FUNCTION_BLOCK FINAL FB_Diagnostics EXTENDS FB_EventLogger 
VAR_IN_OUT
	Control				: ST_System;					  //Machine Control Instance
	Trigger				: BOOL;							  //Diagnostic function call interval
END_VAR
VAR_OUTPUT
	ncpuUsage 			: UDINT;						  //CPU Usage
	nlatency 			: UDINT;						  //CPU Latency
	Outputs 			: ARRAY[0..255] OF ST_Diagnostics;//Devices on ECAT Bus
	ControllerID		: ST_DeviceIdentificationEx;	  //IPC Information
	IPAddress			: T_IPv4Addr;					  //IPC ip address
END_VAR                                                   
VAR                                                       
	_Alarm				: BOOL;							  //Device Alarm
	_AlarmNum			: DINT;							  //Device Alarm Number
	_Warning			: BOOL;							  //Device Warning
	_WarningNum			: DINT;							  //Device Warning Number
	_FaultTimer_ET		: REAL;								//Fault timer elapsed
	_r_Trig				: ARRAY[0..9] OF R_TRIG;    	  //Public Rising Edge Triggers
END_VAR                                                   
VAR_STAT                                                  
	_Masterdata			: ARRAY[0..10] OF ST_Masterdata;  //ECAT Master Device Diagnostic Data
	_DeviceFault		: BOOL;							  //Fault for crc count
	_StatusFault		: BOOL;							  //Fault for status
END_VAR
VAR PERSISTENT          	
	_Name					: STRING[40];				  //Name for HMI
	_Description			: STRING[40];				  //Description for HMI
	_AlarmMute				: BOOL;						  //Alarm Mute
	_FaultTimer_PT			: REAL;						  //Fault timer preset time
END_VAR

M_CPU();
M_Masters();
M_Slaves();
M_AlarmMonitor();
M_AlarmReset();
M_WarningMonitor();

{attribute 'monitoring' := 'variable'}
PROPERTY PUBLIC Alarm : Bool
GET
Alarm := _Alarm;
END_GET
END_PROPERTY

{attribute 'monitoring' := 'variable'}
PROPERTY PUBLIC AlarmMute : BOOL
SET
AlarmMute := _AlarmMute;
END_SET
END_PROPERTY

{attribute 'monitoring' := 'variable'}
PROPERTY PUBLIC Description : String[40]
GET
Description := _Description;
END_GET
SET
_Description := Description;
END_SET
END_PROPERTY

METHOD PRIVATE F_DeviceState_to_String : STRING
VAR_INPUT
	DeviceState: BYTE;
END_VAR
CASE (DeviceState AND 16#0F) OF
	1: F_DeviceState_to_String := 'Init';
	2: F_DeviceState_to_String := 'Pre-Operational';
	3: F_DeviceState_to_String := 'Bootstrap';
	4: F_DeviceState_to_String := 'Safe-Operational';
	8: F_DeviceState_to_String := 'Operational'; 
END_CASE
CASE (DeviceState AND 16#F0) OF
	1: F_DeviceState_to_String := Concat(F_DeviceState_to_String,': Statemachine error in the EtherCAT slave');
	2: F_DeviceState_to_String := Concat(F_DeviceState_to_String,': Invalid VendorId, Product Code, RevisionsNo or SerialNo');
	4: F_DeviceState_to_String := Concat(F_DeviceState_to_String,': Error occured while sending initialization commands.');
END_CASE
RETURN;
END_METHOD

METHOD PRIVATE F_LinkState_to_String : STRING
VAR_INPUT
	LinkState: BYTE;
END_VAR
CASE (LinkState AND 16#0F) OF
	0: F_LinkState_to_String := 'Link status ok';
	1: F_LinkState_to_String := 'No communication with the EtherCAT-Slave';
	2: F_LinkState_to_String := concat(concat('Error at port ', INT_TO_STRING(((LinkState AND 16#F0)/16)-1)), '. The port has a link, but no communication is possible.');
	4: F_LinkState_to_String := concat(concat('Missing link at port ', BYTE_TO_STRING(((LinkState AND 16#F0)/16)-1)), '.');
	8: F_LinkState_to_String := concat(concat('Additional link at port ', BYTE_TO_STRING(((LinkState AND 16#F0)/16)-1)), '.'); 
END_CASE
RETURN;
END_METHOD

{attribute 'monitoring' := 'variable'}
PROPERTY PUBLIC FaultTimer_PT : real
GET
FaultTimer_PT := _FaultTimer_PT;
END_GET
SET
_FaultTimer_PT := FaultTimer_PT;
END_SET
END_PROPERTY

METHOD PRIVATE M_AlarmMonitor
VAR
END_VAR
VAR_INST // added by the converter: edge detectors and wires of the graphical bodies
    _w1, _w2, _w3, _w4, _w5 : BOOL;
END_VAR
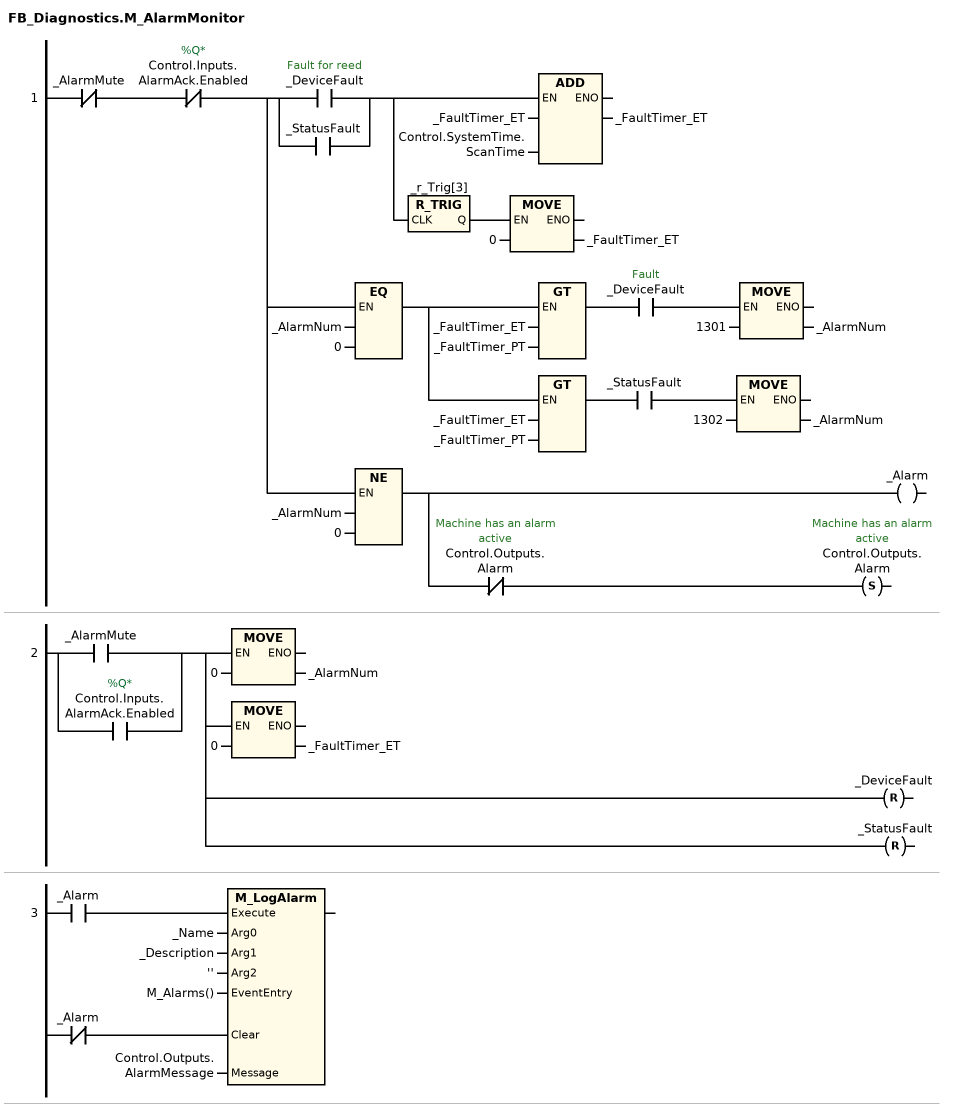
// NETWORK 1
//   Control.Inputs.AlarmAck.Enabled: AT %Q*
//   _DeviceFault: Fault
//   _FaultTimer_ET: Fault timer elapsed
//   Control.SystemTime.ScanTime: Last scan time (Seconds)
//   _FaultTimer_PT: Fault timer preset time
//   Control.Outputs.Alarm: Machine has an alarm active
_w1 := NOT _AlarmMute AND NOT Control.Inputs.AlarmAck.Enabled;
_w2 := _w1 AND (_DeviceFault OR _StatusFault);
IF _w2 THEN _FaultTimer_ET := _FaultTimer_ET + Control.SystemTime.ScanTime; END_IF
_r_Trig[3](CLK := _w2); // R_TRIG
IF _r_Trig[3].Q THEN _FaultTimer_ET := 0; END_IF
_w3 := _w1 AND _AlarmNum = 0;
IF (_w3 AND _FaultTimer_ET > _FaultTimer_PT) AND _DeviceFault THEN _AlarmNum := 1301; END_IF
IF (_w3 AND _FaultTimer_ET > _FaultTimer_PT) AND _StatusFault THEN _AlarmNum := 1302; END_IF
_w4 := _w1 AND _AlarmNum <> 0;
_Alarm := _w4;
Control.Outputs.Alarm S= _w4 AND NOT Control.Outputs.Alarm;

// NETWORK 2
//   Control.Inputs.AlarmAck.Enabled: AT %Q*
//   _FaultTimer_ET: Fault timer elapsed
_w5 := _AlarmMute OR Control.Inputs.AlarmAck.Enabled;
IF _w5 THEN _AlarmNum := 0; END_IF
IF _w5 THEN _FaultTimer_ET := 0; END_IF
_DeviceFault R= _w5;
_StatusFault R= _w5;

// NETWORK 3
M_LogAlarm(Execute := _Alarm, Arg0 := _Name, Arg1 := _Description, Arg2 := '', EventEntry := M_Alarms(), Clear := NOT _Alarm, Message := Control.Outputs.AlarmMessage);
END_METHOD

METHOD PRIVATE M_AlarmReset
VAR_STAT	
	_ClearCRC			:FB_EcMasterFrameStatisticClearCRC; 
	_ClearFrames		:FB_EcMasterFrameStatisticClearFrames;
	_step				: INT;
	_counter			: INT;
END_VAR
// Step engine for resetting etherCat mater errors

CASE _step OF
	0 :	// Initialise and wait for trigger
		_ClearCRC.bExecute:=FALSE;
		_ClearFrames.bExecute:=FALSE;
		_counter := 0;
		IF Control.Inputs.AlarmAck.Enabled THEN _step:=_step+1; END_IF

	
	1 :	// Start getting device ID's 
		_ClearCRC.sNetId := _Masterdata[_counter].NetId;
		_ClearCRC.bExecute:=TRUE;
		IF _ClearCRC.bBusy OR _ClearCRC.bError THEN
		_step:=_step+1; END_IF

	
	2 :	// Getting ID's complete
		_ClearCRC.bExecute:=FALSE;
		IF NOT _ClearCRC.bBusy THEN
		_step:=_step+1;END_IF

	
	3 :	// Start getting device name from device ID
		_ClearFrames.sNetId := _Masterdata[_counter].NetId;
		_ClearFrames.bExecute:=TRUE;
		IF _ClearFrames.bBusy OR _ClearFrames.bError THEN
		_step:=_step+1;END_IF

	
	4 :	// Getting device name complete
		_ClearFrames.bExecute:=FALSE;
		IF NOT _ClearFrames.bBusy THEN
		_step:=_step+1;END_IF

		
	5 :	// Start getting device AMS Net ID from device ID
		_counter := _counter + 1;
		IF _counter >= 11 THEN
		_step:=0;ELSE
		_step:=1;END_IF
			
ELSE
	_step:=0;
END_CASE

// Function block calls
_ClearCRC(sNetId:=);
_ClearFrames(sNetId:=);
END_METHOD

METHOD M_Alarms : TcEventEntry
VAR_INPUT
END_VAR
CASE _AlarmNum OF
	1301: M_Alarms:= TC_Events.TcDiagnostics.A_1301;//Module Fault	
	1302: M_Alarms:= TC_Events.TcDiagnostics.A_1302;//Status Fault			
ELSE
	M_Alarms:= TC_Events.TcDiagnostics.A_Undefined;
END_CASE
END_METHOD

METHOD M_CPU
VAR_STAT
	_DeviceInfo			: FB_GetDeviceIdentificationEx;
	_HostAddr			: FB_GetHostAddrByName;
	_cpuUsage			: TC_CpuUsage;
	_latency			: TC_SysLatency;	
	_incrementer		: INT;	
	_step				: INT;
END_VAR
// Step engine for reading cpu info and status

CASE _step OF
	0 :	// Initialise
		_DeviceInfo.bExecute := FALSE;
		_HostAddr.bExecute := FALSE;
		_cpuUsage.START := FALSE;
		_latency.START := FALSE;
		_step:=_step+1;

	
	1 :	// Start getting device info
		_DeviceInfo.bExecute := TRUE;
		IF _DeviceInfo.bBusy THEN
		_step:=_step+1; END_IF

	
	2 :	// Getting device info completed
		_DeviceInfo.bExecute := FALSE;
		IF NOT _DeviceInfo.bBusy THEN
		_step:=_step+1; END_IF

	
	3 :	// Start getting host AMS address
		_HostAddr.bExecute := TRUE;
		IF _HostAddr.bBusy THEN
		_step:=_step+1; END_IF

	
	4 :	// Getting host AMS address completed
		_HostAddr.bExecute := FALSE;
		IF NOT _HostAddr.bBusy THEN
		_step:=_step+1; END_IF

		
	5 :	// Update outputs
		ControllerID := _DeviceInfo.stDevIdent;
		IPAddress := _HostAddr.sAddr;
		_step:=_step+1;

	
	6 :	// Wait for update trigger
		IF Trigger THEN _step:=_step+1; END_IF

	
	7: 	// Read the cpu usage
		_cpuUsage.START := TRUE;
		IF _cpuUsage.BUSY THEN
		_step:=_step+1; END_IF

		
	8:	// Cpu usage read complete
		_cpuUsage.START := FALSE;
		IF NOT _cpuUsage.BUSY THEN
		_step:=_step+1; END_IF
		
	9:	// Read cpu latency
		_latency.START := TRUE;
		IF _latency.BUSY THEN
		_step:=_step+1; END_IF

		
	10:	// Cpu latency read complete
		_latency.START := FALSE;
		IF NOT _latency.BUSY THEN
		_step:=_step+1; END_IF

		
	11:	// Update outputs and go back to waiting for trigger
		ncpuUsage := _cpuUsage.USAGE;
		nlatency := _latency.ACTUAL;
		_step:=6;
		
ELSE
	_step:=0;
END_CASE

// Function block calls
_DeviceInfo();
_HostAddr(sNetID:=ControllerID.strAmsNetId);
_cpuUsage(NETID:=ControllerID.strAmsNetId);
_latency(NETID:=ControllerID.strAmsNetId);
END_METHOD

METHOD PRIVATE M_Masters
VAR_STAT
	_GetDeviceIDs 				: IOF_GetDeviceIDs;
	_IdsData             		: ARRAY[0..10] OF WORD;	
	_GetDeviceName 				: IOF_GetDeviceName;
	_GetDeviceNetId 			: IOF_GetDeviceNetId;	
	_EcMasterFrameStatistic		: FB_EcMasterFrameStatistic; 
	_GetMasterState    			: FB_EcGetMasterState;
	_step						: INT;
	_counter					: INT;
END_VAR
// Step engine for retrieving etherCat mater info and status
CASE _step OF
	0 :	// Initialise and wait for trigger
		_GetDeviceIDs.START:=FALSE;
		_GetDeviceName.START:=FALSE;
		_GetDeviceNetId.START:=FALSE;
		_EcMasterFrameStatistic.bExecute:=FALSE;
		_GetMasterState.bExecute:=FALSE;
		_counter := 0;
		IF Trigger THEN _step:=_step+1; END_IF
	
	1 :	// Start getting device ID's 
		_GetDeviceIDs.START:=TRUE;
		IF _GetDeviceIDs.BUSY OR _GetDeviceIDs.ERR THEN
		_step:=_step+1; END_IF

	2 :	// Getting ID's complete
		_GetDeviceIDs.START:=FALSE;
		IF NOT _GetDeviceIDs.BUSY THEN
		_step:=_step+1;END_IF
	
	3 :	// Start getting device name from device ID
		_GetDeviceName.DEVICEID := _IdsData[_counter+1];
		_GetDeviceName.START:=TRUE;
		IF _GetDeviceName.BUSY OR _GetDeviceName.ERR THEN
		_step:=_step+1;END_IF
	
	4 :	// Getting device name complete
		_GetDeviceName.START:=FALSE;
		IF NOT _GetDeviceName.BUSY THEN
		_step:=_step+1;END_IF
	
	5 :	// Start getting device AMS Net ID from device ID
		_GetDeviceNetId.DEVICEID := _IdsData[_counter+1];
		_GetDeviceNetId.START:=TRUE;
		IF _GetDeviceNetId.BUSY OR _GetDeviceNetId.ERR THEN
		_step:=_step+1;END_IF
	
	6 :	// Getting device AMS Net ID complete
		_GetDeviceNetId.START:=FALSE;
		IF NOT _GetDeviceNetId.BUSY THEN
		_step:=_step+1;END_IF

	7: 	// Start getting master frame statistics from AMS Net ID
		_EcMasterFrameStatistic.sNetId := _GetDeviceNetId.DeviceNetId;
		_EcMasterFrameStatistic.bExecute := TRUE;
		IF _EcMasterFrameStatistic.bBusy OR _EcMasterFrameStatistic.bError THEN 
		_step := _step+1; END_IF
		
	8:	// Getting frame statistics complete
		_EcMasterFrameStatistic.bExecute:=FALSE;
		IF NOT _EcMasterFrameStatistic.bBusy THEN 
			_step := _step+1; 
		END_IF
	
	9:	// Start getting master status from AMS Net ID
		_GetMasterState.sNetId := _GetDeviceNetId.DeviceNetId;
		_GetMasterState.bExecute := TRUE;
		IF _GetMasterState.bBusy OR _GetMasterState.bError THEN 
		_step := _step+1; END_IF
		
	10:	// Getting master status complete
		IF NOT _GetMasterState.bBusy THEN 
			_GetMasterState.bExecute:=FALSE;
			_step := _step+1; 
		END_IF
	
	11:	// Update master data array
		_Masterdata[_counter].ID := _IdsData[_counter+1];
		_Masterdata[_counter].Name := _GetDeviceName.DEVICENAME;
		_Masterdata[_counter].NetId := _GetDeviceNetId.DeviceNetId;
		_Masterdata[_counter].FramesPerSecond := _EcMasterFrameStatistic.fFramesPerSecond;
		_Masterdata[_counter].LostFrames := _EcMasterFrameStatistic.nLostFrames;
		_Masterdata[_counter].LostQueuedFrames := _EcMasterFrameStatistic.nLostQueuedFrames;
		_Masterdata[_counter].QueuedFramesPerSecond := _EcMasterFrameStatistic.fQueuedFramesPerSecond;
		
		// Convert state word to status text
		IF    _GetMasterState.state = 1 THEN _Masterdata[_counter].Status := 'Init';
		ELSIF _GetMasterState.state = 2 THEN _Masterdata[_counter].Status := 'Pre-Operational';
		ELSIF _GetMasterState.state = 4 THEN _Masterdata[_counter].Status := 'Safe-Operational';
		ELSIF _GetMasterState.state = 8 THEN _Masterdata[_counter].Status := 'Operational';
		ELSE _Masterdata[_counter].Status := 'unknown'; END_IF
		_counter := _counter + 1;
		
		// If another master is in list then retrieve details or return to start and wait for trigger
		IF _IdsData[_counter+1] > 0 THEN
			_step:=3;
		ELSE
			_counter := 0;
			_step:=0;
		END_IF		
ELSE
	_step:=0;
END_CASE

// Function block calls
_GetDeviceIDs(NETID:=,LEN:=SIZEOF(_IdsData),DESTADDR:=ADR(_IdsData));
_GetDeviceName(NETID:=);
_GetDeviceNetId(NETID:=);
_EcMasterFrameStatistic(); 
_GetMasterState();
END_METHOD

METHOD PRIVATE M_Slaves
VAR_STAT
	_step					: INT;
	_counter				: INT;
	_pntr					: INT;
	_MasterCounter			: INT;
	_GetConfSlaves			: FB_EcGetConfSlaves;
	_GetAllSlaveCrcErrors	: FB_EcGetAllSlaveCrcErrors;
	_GetAllSlaveStates		: FB_EcGetAllSlaveStates;
	_crcErrors              : ARRAY[0..255] OF DWORD; 
	_Configs           		: ARRAY[0..255] OF ST_EcSlaveConfigData; 
    _devStates           	: ARRAY[0..255] OF ST_EcSlaveState; 
END_VAR
// Step engine to retrieve etherCat slave device info and status
CASE _step OF
	0 :	// Initialise and wait for trigger
		_GetConfSlaves.bExecute:= FALSE;
		_GetAllSlaveStates.bExecute:= FALSE;
		_GetAllSlaveCrcErrors.bExecute:= FALSE;
		_pntr := 0;
		_counter := 0;
		_MasterCounter := 0;
		IF Trigger THEN _step:=_step+1; END_IF

	1:	// Get master data for output array
		Outputs[_pntr].Name := _Masterdata[_MasterCounter].Name;
		Outputs[_pntr].Address := _Masterdata[_MasterCounter].ID;
		Outputs[_pntr].LostFrames := _Masterdata[_MasterCounter].LostFrames;
		Outputs[_pntr].FramesPerSecond := _Masterdata[_MasterCounter].FramesPerSecond;
		Outputs[_pntr].LostQueuedFrames := _Masterdata[_MasterCounter].LostQueuedFrames;
		Outputs[_pntr].QueuedFramesPerSecond := _Masterdata[_MasterCounter].QueuedFramesPerSecond;
		Outputs[_pntr].NetId := _Masterdata[_MasterCounter].NetId;
		Outputs[_pntr].DeviceStatus := _Masterdata[_MasterCounter].Status;
		_pntr := _pntr + 1;
		
		// Set device and status alarms
		IF _GetAllSlaveStates.nSlaves > 0 THEN
			IF Outputs[_pntr].LostQueuedFrames > 0 OR Outputs[_pntr].LostFrames > 0THEN 
				_Name := Outputs[_pntr].Name;
				_Description := concat(concat('Lost ',UDINT_TO_STRING(Outputs[_pntr].LostFrames + Outputs[_pntr].LostQueuedFrames)),' frames.');
				_DeviceFault := TRUE;
			END_IF
			IF Outputs[_pntr].DeviceStatus <> 'Operational' THEN
				_Name := Outputs[_pntr].Name;
				_Description := Outputs[_pntr].DeviceStatus;
				_StatusFault := TRUE; 
			END_IF
		END_IF
		
		_step:=_step+1;
	2:	// Start getting slave configurations for selected master
		_GetConfSlaves.sNetId:=_Masterdata[_MasterCounter].NetId;
		_GetConfSlaves.bExecute:= TRUE;
		IF _GetConfSlaves.bBusy OR _GetConfSlaves.bError THEN
		_step:=_step+1; END_IF

	3:	// Getting slave configurations complete
		_GetConfSlaves.bExecute:= FALSE;
		IF NOT _GetConfSlaves.bBusy THEN
		_step:=_step+1; END_IF
	
	4:	// Start getting slave crc errors for selected master
		_GetAllSlaveCrcErrors.sNetId:=_Masterdata[_MasterCounter].NetId;
		_GetAllSlaveCrcErrors.bExecute:= TRUE;
		IF _GetAllSlaveCrcErrors.bBusy OR _GetAllSlaveCrcErrors.bError THEN
		_step:=_step+1; END_IF

	
	5:	// Getting slave crc errors complete
		_GetAllSlaveCrcErrors.bExecute:= FALSE;
		IF NOT _GetAllSlaveCrcErrors.bBusy THEN
		_step:=_step+1; END_IF

	6: 	// Start getting slave states for selected master
		_GetAllSlaveStates.sNetId:=_Masterdata[_MasterCounter].NetId;
		_GetAllSlaveStates.bExecute:= TRUE;
		IF _GetAllSlaveStates.bBusy OR _GetAllSlaveStates.bError THEN
		_step:=_step+1; END_IF

	7:	// Getting slave states complete
		_GetAllSlaveStates.bExecute:= FALSE;
		IF NOT _GetAllSlaveStates.bBusy THEN
		_step:=_step+1; END_IF
	
	8:	// Update output array with all slaves for selected master
		IF _GetAllSlaveStates.nSlaves > 0 THEN
			FOR _counter := 0 TO UINT_TO_INT(_GetAllSlaveStates.nSlaves-1) BY 1 DO
				
				Outputs[_pntr].Name := _Configs[_counter].sName;
				Outputs[_pntr].ProductType := _Configs[_counter].sType;
				Outputs[_pntr].CRCError := _crcErrors[_counter];
				Outputs[_pntr].Address := _Configs[_counter].nAddr;
				Outputs[_pntr].LinkStatus := F_LinkState_to_String(_Configs[_counter].nLinkStatus);
				Outputs[_pntr].DeviceStatus := F_DeviceState_to_String(_devStates[_counter].deviceState);
				Outputs[_pntr].NetId := '';
				
				// Set device and status alarms
				IF Outputs[_pntr].CRCError > 0 THEN 
					_Name := Outputs[_pntr].Name;
					_Description := concat(DWORD_TO_STRING(Outputs[_pntr].CRCError),' CRC Errors.');
					_DeviceFault := TRUE; 
				END_IF
				IF Outputs[_pntr].DeviceStatus <> 'Operational' OR Outputs[_pntr].LinkStatus <> 'Link status ok' THEN 
					_Name := Outputs[_pntr].Name;
					_Description := Outputs[_pntr].DeviceStatus;
					_StatusFault := TRUE; 
				END_IF
				
				_pntr := _pntr + 1;
				
			END_FOR
		END_IF
		_step:=_step+1;
	
	9:	// Check if another master in cue and repeat sequence or step forward
		_MasterCounter:=_MasterCounter+1;
		IF _Masterdata[_MasterCounter].Name = '' THEN
		_step:=_step+1; ELSE _step:=1; END_IF	
	
	10:	// Clear the remainder of the output array
		FOR _counter := _pntr TO 255 BY 1 DO
			
			Outputs[_counter].Name := '';
			Outputs[_counter].ProductType := '';
			Outputs[_counter].CRCError := 0;
			Outputs[_counter].Address := 0;
			Outputs[_counter].LinkStatus := '';
			Outputs[_counter].DeviceStatus := '';
			
		END_FOR
		_step:=0;
		
ELSE
	_step:=0;
END_CASE

// Function block calls
_GetConfSlaves(pArrEcConfSlaveInfo := ADR(_Configs), cbBufLen:= SIZEOF(_Configs));
_GetAllSlaveStates(pStateBuf := ADR(_devStates), cbBufLen:=SIZEOF(_devStates));
_GetAllSlaveCrcErrors(pCrcErrorBuf := ADR(_crcErrors), cbBufLen:= SIZEOF(_crcErrors));
END_METHOD

METHOD PRIVATE M_WarningMonitor
VAR_INPUT
END_VAR
VAR_INST
END_VAR
VAR_INST // added by the converter: edge detectors and wires of the graphical bodies
    _w1 : BOOL;
END_VAR
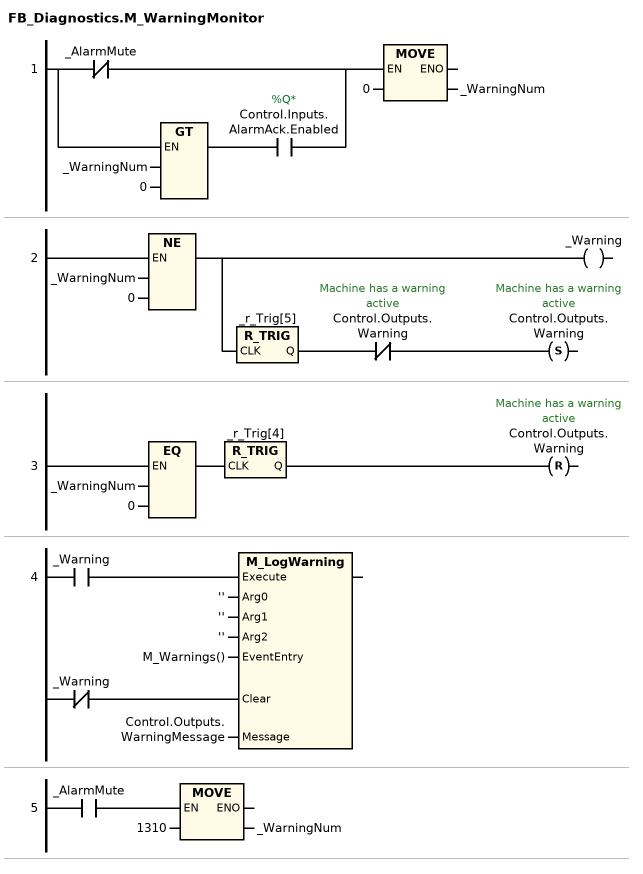
// NETWORK 1
//   Control.Inputs.AlarmAck.Enabled: AT %Q*
IF NOT _AlarmMute OR _WarningNum > 0 AND Control.Inputs.AlarmAck.Enabled THEN _WarningNum := 0; END_IF

// NETWORK 2
//   Control.Outputs.Warning: Machine has a warning active
_w1 := _WarningNum <> 0;
_Warning := _w1;
_r_Trig[5](CLK := _w1); // R_TRIG
Control.Outputs.Warning S= _r_Trig[5].Q AND NOT Control.Outputs.Warning;

// NETWORK 3
//   Control.Outputs.Warning: Machine has a warning active
_r_Trig[4](CLK := _WarningNum = 0); // R_TRIG
Control.Outputs.Warning R= _r_Trig[4].Q;

// NETWORK 4
M_LogWarning(Execute := _Warning, Arg0 := '', Arg1 := '', Arg2 := '', EventEntry := M_Warnings(), Clear := NOT _Warning, Message := Control.Outputs.WarningMessage);

// NETWORK 5
IF _AlarmMute THEN _WarningNum := 1310; END_IF
END_METHOD

METHOD M_Warnings : TcEventEntry
VAR_INPUT
END_VAR
CASE _WarningNum OF
	1310: M_Warnings:= TC_Events.TcDiagnostics.W_1310;//Alarm Mute Active					
ELSE
	M_Warnings:=  TC_Events.TcDiagnostics.W_Undefined;	
END_CASE
END_METHOD

{attribute 'monitoring' := 'variable'}
PROPERTY PUBLIC Name : String[40]
GET
Name := _Name;
END_GET
SET
_Name := Name;
END_SET
END_PROPERTY

{attribute 'monitoring' := 'variable'}
PROPERTY PUBLIC Warning : Bool
GET
Warning := _Warning;
END_GET
END_PROPERTY

END_FUNCTION_BLOCK

(* stored: Version 1.1.0.1, ProductVersion 3.1.4024.3
   POU FB_Diagnostics: Id {6a3a25e4-3108-4d31-894c-fbeac9d0dec1}, SpecialFunc None
   Property Alarm: Id {69110e00-4523-4fa9-89d0-50ae4bf20a84}
   Get Get: Id {8bc6c785-497f-40c8-bc2b-986760db2081}
   Property AlarmMute: Id {63a0c7ea-2df5-4b89-b784-e4e099473d5d}
   Set Set: Id {ab8b9816-b635-4a65-b94b-1bb65680ec39}
   Property Description: Id {96797581-e9e8-4b48-8e24-c3e537d32b54}
   Get Get: Id {7923df63-1841-47e7-b74a-c288695c9364}
   Set Set: Id {db7a416c-199b-4d4a-b112-c8356822c2da}
   Method F_DeviceState_to_String: Id {682e0877-2bce-47d5-a239-0bb40247fa6b}
   Method F_LinkState_to_String: Id {f36ff1f5-3f55-462b-ad0c-5b028b0fa95d}
   Property FaultTimer_PT: Id {deccdbaa-55a0-47bc-a96a-b98e24452847}
   Get Get: Id {3261280c-54c7-4fc2-a17a-3e2023038257}
   Set Set: Id {97af4c69-17d7-4d52-bbcb-78e9e6fd2135}
   Method M_AlarmMonitor: Id {8b4b1cc8-ac65-4e81-96e3-63e9ab17f9b0}
   Method M_AlarmReset: Id {2cff5ebe-d38f-4fe2-943d-b12b7a0f4b99}
   Method M_Alarms: Id {2359c73b-2093-4c22-8bfb-0cb83d48160d}
   Method M_CPU: Id {55a330b9-c115-461a-9541-f2993f7e681f}
   Method M_Masters: Id {da8d987c-8e96-4367-ac07-405993ce6181}
   Method M_Slaves: Id {d6863cba-c367-4740-8fb3-59c73c3a6474}
   Method M_WarningMonitor: Id {54cf49d2-0ffb-42dd-bdb1-23040bdc620b}
   Method M_Warnings: Id {a1382a26-8d98-4175-9387-eb65a2dd80ab}
   Property Name: Id {c694a9c1-da00-4d1d-98ec-c0e230801529}
   Get Get: Id {a5d13d54-68c9-4a01-b369-844af918b5e7}
   Set Set: Id {64b2ab2f-3f53-4fb6-80c8-422e9b01a55e}
   Property Warning: Id {514172d3-d1a7-4c87-8611-e4925a96cabb}
   Get Get: Id {5623ddc0-c5a8-4f7a-9841-5a81ee6d2bb8} *)
